// TIA Portal project "WEB" (V14)

(* hardware
DEVICE "S71500/ET200MP station_1"  S7-1500 station
   slot 0: "Rail_0"  Rack  6ES7 590-1***0-0AA0
   slot 1: "PLC_1"  CPU 1516F-3 PN/DP  6ES7 516-3FN01-0AB0  V2.0
      slot 3: "CPU display_1"  6ES7591-1BA00-0AA0
*)

// ===== PLC "PLC_1"  CPU 1516F-3 PN/DP =====

DATA_BLOCK "Main_Safety_RTG1_DB"   // DB1, F_DB
{ S7_Optimized_Access := 'TRUE' }
NAME : FUSI
VERSION : 0.1
// stored: InstanceOfName Main_Safety_RTG1
"Main_Safety_RTG1"
BEGIN
END_DATA_BLOCK

DATA_BLOCK "Regulator 1"   // DB2
TITLE = Regulator1
{ S7_Optimized_Access := 'TRUE' }
VERSION : 0.1
   VAR
      c : Real := 3.0E+08;
      theAnswer : Int := 55;
      h : Real := 7.626;
      pi : Real := 3.141593;
      g : Real := 9.81;
      enable : Bool := true;
      auto : Bool := 1;
   END_VAR
BEGIN
END_DATA_BLOCK

DATA_BLOCK "Regulator 2"   // DB3
TITLE = Regulator1
{ S7_Optimized_Access := 'TRUE' }
VERSION : 0.1
   VAR
      c : Real := 3.0E+08;
      theAnswer : Real := 42.0;
      h : Real := 6.626;
      pi : Real := 3.141593;
      g : Real := 9.81;
      enable : Bool := true;
      auto : Bool := false;
   END_VAR
BEGIN
END_DATA_BLOCK

DATA_BLOCK "Analog Output 1"   // DB4
TITLE = Regulator1
{ S7_Optimized_Access := 'TRUE' }
VERSION : 0.1
   VAR
      c : Real := 3.0E+08;
      theAnswer : Int := 55;
      h : Real := 7.626;
      pi : Real := 3.141593;
      g : Real := 9.81;
      enable : Bool := true;
      auto : Bool := 1;
   END_VAR
BEGIN
END_DATA_BLOCK

DATA_BLOCK "Analog Input 1"   // DB5
TITLE = Regulator1
{ S7_Optimized_Access := 'TRUE' }
VERSION : 0.1
   VAR
      c : Real := 3.0E+08;
      theAnswer : Int := 55;
      h : Real := 7.626;
      pi : Real := 3.141593;
      g : Real := 9.81;
      enable : Bool := true;
      auto : Bool := 1;
   END_VAR
BEGIN
END_DATA_BLOCK

DATA_BLOCK "Diameter Calculation 1"   // DB6
TITLE = Regulator1
{ S7_Optimized_Access := 'TRUE' }
VERSION : 0.1
   VAR
      c : Real := 3.0E+08;
      theAnswer : Int := 55;
      h : Real := 7.626;
      pi : Real := 3.141593;
      g : Real := 9.81;
      enable : Bool := true;
      auto : Bool := 1;
   END_VAR
BEGIN
END_DATA_BLOCK

DATA_BLOCK "Diameter Calculation 2"   // DB7
TITLE = Regulator1
{ S7_Optimized_Access := 'TRUE' }
VERSION : 0.1
   VAR
      c : Real := 3.0E+08;
      theAnswer : Real := 42.0;
      h : Real := 6.626;
      pi : Real := 3.141593;
      g : Real := 9.81;
      enable : Bool := true;
      auto : Bool := false;
   END_VAR
BEGIN
END_DATA_BLOCK

DATA_BLOCK "Analog Output 2"   // DB8
TITLE = Regulator1
{ S7_Optimized_Access := 'TRUE' }
VERSION : 0.1
   VAR
      c : Real := 3.0E+08;
      theAnswer : Real := 42.0;
      h : Real := 6.626;
      pi : Real := 3.141593;
      g : Real := 9.81;
      enable : Bool := true;
      auto : Bool := false;
   END_VAR
BEGIN
END_DATA_BLOCK

DATA_BLOCK "Analog Input 2"   // DB9
TITLE = Regulator1
{ S7_Optimized_Access := 'TRUE' }
VERSION : 0.1
   VAR
      c : Real := 3.0E+08;
      theAnswer : Real := 42.0;
      h : Real := 6.626;
      pi : Real := 3.141593;
      g : Real := 9.81;
      enable : Bool := true;
      auto : Bool := false;
   END_VAR
BEGIN
END_DATA_BLOCK

FUNCTION_BLOCK "Main_Safety_RTG1"   // FB1, F_FBD
{ S7_Optimized_Access := 'TRUE' }
VERSION : 0.1
BEGIN
END_FUNCTION_BLOCK

ORGANIZATION_BLOCK "Main"   // OB1, LAD, ProgramCycle
TITLE = "Main Program Sweep (Cycle)"
{ S7_Optimized_Access := 'TRUE' }
VERSION : 0.1
   VAR_INPUT
      Initial_Call : Bool;   // Initial call of this OB
      Remanence : Bool;   // =True, if remanent data are available
   END_VAR
   VAR_TEMP
      Ret : Int;
   END_VAR
BEGIN

REGION Network 1
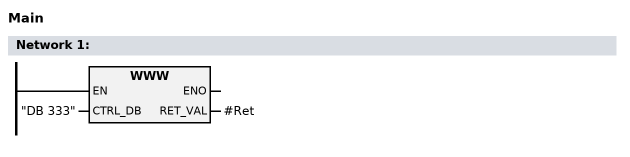
   #Ret := WWW(CTRL_DB := "DB 333");
END_REGION
END_ORGANIZATION_BLOCK